(* PLC project Unnamed, Unknown Unnamed 1 *)
(* stored: creationDateTime 2026-06-15T08:02:50, modificationDateTime 2026-06-15T08:02:50 *)

FUNCTION MK_PTR : __XWORD
  VAR_INPUT
    IN : ANY;
  END_VAR

END_FUNCTION

PROGRAM PLC_PRG
  VAR
    src : INT;
    p : POINTER TO INT;
  END_VAR

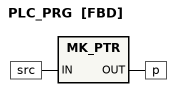
(* FBD diagram, written out as Structured Text *)
p := MK_PTR(src);
END_PROGRAM

CONFIGURATION Config0
  RESOURCE Res0 ON PLC
    TASK task0(INTERVAL := T#20ms, PRIORITY := 1);
    PROGRAM instance0 WITH task0 : PLC_PRG;
  END_RESOURCE
END_CONFIGURATION
